{attribute 'linkalways'} 
{attribute 'no_explicit_call' := 'This FB is a CLASS and must be accessed using methods or properties'}
{attribute 'enable_dynamic_creation'}
FUNCTION_BLOCK _ETcVnPixelConnectivity EXTENDS EnumDatatypeBase
VAR
	localData : ETcVnPixelConnectivity;
	activeData : REFERENCE TO ETcVnPixelConnectivity;
	enumBaseDatatype : _DINT(localData);
END_VAR

METHOD PRIVATE AddLocalEnumeration
VAR_INPUT
	Enumeration : T_MAXSTRING;
	Value : ETcVnPixelConnectivity;
END_VAR
AddEnumeration(Enumeration, Value);
END_METHOD

PROPERTY PUBLIC Address : PVOID
GET
Address := ADR(activeData);
END_GET
END_PROPERTY

METHOD PUBLIC ClearReference
VAR_INPUT
END_VAR
activeData REF= localData;
SetBaseDatatypeReference();
END_METHOD

METHOD PUBLIC Clone : I_Datatype
VAR
    pClone : POINTER TO _ETcVnPixelConnectivity;
END_VAR
pClone := __NEW(_ETcVnPixelConnectivity(InitialValue := Value));
Clone := pClone^;
END_METHOD

METHOD FB_init : BOOL
VAR_INPUT
	bInitRetains : BOOL; // if TRUE, the retain variables are initialized (warm start / cold start)
	bInCopyCode : BOOL;  // if TRUE, the instance afterwards gets moved into the copy code (online change)
	InitialValue : ETcVnPixelConnectivity;
END_VAR
localData := InitialValue;
AddBaseDatatype(enumBaseDatatype);
ClearReference();

AddLocalEnumeration('TCVN_PC_4', ETcVnPixelConnectivity.TCVN_PC_4);
AddLocalEnumeration('TCVN_PC_8', ETcVnPixelConnectivity.TCVN_PC_8);
END_METHOD

PROPERTY PUBLIC Identifier : T_MAXSTRING
GET
Identifier := 'ETcVnPixelConnectivity';
END_GET
END_PROPERTY

METHOD IsEnumeratorValueEqual : BOOL
VAR_INPUT
	Enumerator : I_KeyValueForwardEnumerator;
END_VAR
VAR
	storedValue : ETcVnPixelConnectivity;
END_VAR
IF NOT Enumerator.TryGet(storedValue) THEN
	RETURN;
END_IF

IsEnumeratorValueEqual := storedValue = activeData;
END_METHOD

METHOD PUBLIC MakeReferenceTo
VAR_INPUT
	ReferenceTarget : REFERENCE TO ETcVnPixelConnectivity;
END_VAR
activeData REF= ReferenceTarget;
SetBaseDatatypeReference();
END_METHOD

METHOD PROTECTED SetBaseDatatypeReference
VAR_INPUT
END_VAR
enumBaseDatatype.MakeReferenceTo(activeData);
END_METHOD

PROPERTY PUBLIC Size : UDINT
GET
Size := SIZEOF(activeData);
END_GET
END_PROPERTY

METHOD TryMakeReferenceTo : BOOL
VAR_INPUT
	Target : I_Datatype;
END_VAR
VAR
	pTargetData : POINTER TO ETcVnPixelConnectivity;
END_VAR
IF NOT IsEquivalentTo(Target) THEN
	RETURN;
END_IF

pTargetData := Target.Address;
activeData REF= pTargetData^;
SetBaseDatatypeReference();
TryMakeReferenceTo := TRUE;
END_METHOD

PROPERTY PUBLIC Value : ETcVnPixelConnectivity
GET
Value := activeData;
END_GET
SET
activeData := Value;
END_SET
END_PROPERTY

END_FUNCTION_BLOCK

(* stored: Version 1.1.0.1, ProductVersion 3.1.4024.13
   POU _ETcVnPixelConnectivity: Id {00d7e4fe-0919-0d89-1765-aec693ce9d92}, SpecialFunc None
   Folder Core: Id {71348b75-451f-08ad-2e6b-f1b9c3e99389}
   Folder Protected: Id {8615825c-9473-08c7-3270-a2c8e31de5a3}
   Folder Customize: Id {f1bc5966-599f-0aa9-2261-7baceea11227}
   Folder Constructor: Id {208f36ac-7f83-027b-13cf-fddb87a340f2}
   Folder Private: Id {7478ad53-ff7d-015a-1ce5-03f65c107ed9}
   Folder Protected: Id {8eee0925-cc27-0b3c-234c-7a2344437599}
   Method AddLocalEnumeration: Id {611aed11-379c-02da-3c15-21d9f424bae9}
   Property Address: Id {66098a22-4cf4-0f51-1134-55eb4303bb0b}
   Get Get: Id {786a031d-a731-0e10-0caf-6d43249dbd12}
   Method ClearReference: Id {cec4f0b3-7d91-01da-1663-f3b94987bfc0}
   Method Clone: Id {2cd5d6a7-9217-05df-00c8-7273226e0161}
   Method FB_init: Id {718405cb-445a-0e58-2a6e-4f98b4dfa2a7}
   Property Identifier: Id {347a1130-88a6-057f-1979-4f27431e1aa0}
   Get Get: Id {91426f67-ca7a-0e58-3686-aa2f7b19d417}
   Method IsEnumeratorValueEqual: Id {87ca2e3a-62af-01fe-0e2b-e7914c6e85d7}
   Method MakeReferenceTo: Id {24625d42-60b3-0202-3ff9-9b20aa2d7c8b}
   Method SetBaseDatatypeReference: Id {3e62b2f7-d6f4-00d6-098e-64214e655acc}
   Property Size: Id {a8d45146-d613-0670-0e65-9ccec660594a}
   Get Get: Id {8beeed32-0f74-03d9-0b5a-e845852aa775}
   Method TryMakeReferenceTo: Id {6906f907-d4b7-03bf-08fb-b89b17d834d7}
   Property Value: Id {71f06e9d-9e8d-0c0a-3369-6878f6f03e1f}
   Get Get: Id {d56f4e0b-7a24-0ae8-3e9e-6e0e38518a1b}
   Set Set: Id {08e1d0c1-92ed-0a9a-2d3f-415274f016ab} *)
